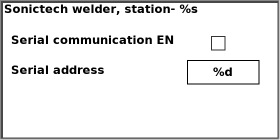
VISUALIZATION vSonicTechSet  // 280x140
VAR_IN_OUT
	stData:stSonicTech_MachSettings;
END_VAR
VAR_INPUT
	sName:STRING;
END_VAR
    Rectangle (1,1 278x138), "Sonictech welder, station- %s", text variable: sName
    Rectangle (187,60 72x24), "%d", text variable: stData.bySerialAdress
        OnMouseDown: write the text variable via Default, min 1, max 128, title 'RS485 Fildbus address', format %d
    Label (8,60 180x20), "Serial address"
    Label (8,30 180x20), "Serial communication EN"
    Checkbox (209,30 26x26), variable: stData.bSerialCommunicationEN
END_VISUALIZATION

(* stored: Version 1.1.0.1, ProductVersion 3.1.4024.13
   Visu vSonicTechSet: Id {51ec0da9-248a-4041-9973-306cfad667b3} *)
